// Mitsubishi GX Works2 project: k10   PLC: Q02/Q02H

PROGRAM MAIN
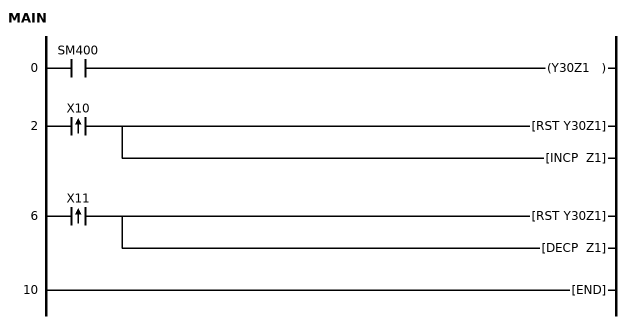
0     LD      SM400
      OUT     Y30Z1
2     LDP     X10
      RST     Y30Z1
      INCP    Z1
6     LDP     X11
      RST     Y30Z1
      DECP    Z1
10    END
END_PROGRAM
